% RSLogix 500 project Hourmeter.RSS, saved by version 8.30.00.16 %
PROJECT "UNTITLED"    % processor: Bul.1763 MicroLogix 1100 Series B %

PROGRAM FILES
  LAD 2   11 rungs

DATA FILES
  O0 OUTPUT  4 elements
  I1 INPUT  6 elements
  S2 STATUS  66 elements
  B3 BINARY  1 elements
  T4 TIMER  1 elements
  C5 COUNTER  3 elements
  R6 CONTROL  1 elements
  N7 INTEGER  5 elements
  F8 FLOAT  1 elements

LADDER 2
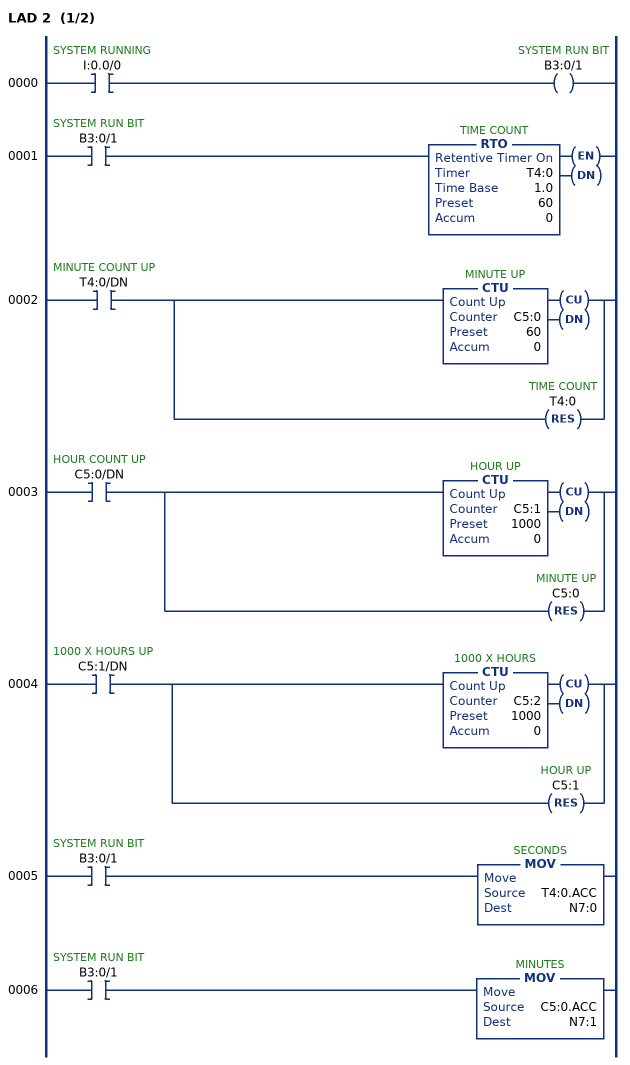
% Rung: 0 %
SOR XIC I:0.0/0 OTE B3:0/1 EOR
%   I:0.0/0  "SYSTEM RUNNING" %
%   B3:0/1  "SYSTEM RUN BIT" %
% Rung: 1 %
SOR XIC B3:0/1 RTO T4:0 1.0 60 0 EOR
%   B3:0/1  "SYSTEM RUN BIT" %
%   T4:0  "TIME COUNT" %
% Rung: 2 %
SOR XIC T4:0/DN BST CTU C5:0 60 0 NXB RES T4:0 BND EOR
%   T4:0/DN  "MINUTE COUNT UP" %
%   C5:0  "MINUTE UP" %
%   T4:0  "TIME COUNT" %
% Rung: 3 %
SOR XIC C5:0/DN BST CTU C5:1 1000 0 NXB RES C5:0 BND EOR
%   C5:0/DN  "HOUR COUNT UP" %
%   C5:1  "HOUR UP" %
%   C5:0  "MINUTE UP" %
% Rung: 4 %
SOR XIC C5:1/DN BST CTU C5:2 1000 0 NXB RES C5:1 BND EOR
%   C5:1/DN  "1000 X HOURS UP" %
%   C5:2  "1000 X HOURS" %
%   C5:1  "HOUR UP" %
% Rung: 5 %
SOR XIC B3:0/1 MOV T4:0.ACC N7:0 EOR
%   B3:0/1  "SYSTEM RUN BIT" %
%   T4:0.ACC  "SECONDS" %
%   N7:0  "SECONDS" %
% Rung: 6 %
SOR XIC B3:0/1 MOV C5:0.ACC N7:1 EOR
%   B3:0/1  "SYSTEM RUN BIT" %
%   C5:0.ACC  "MINUTES" %
%   N7:1  "MINUTES" %

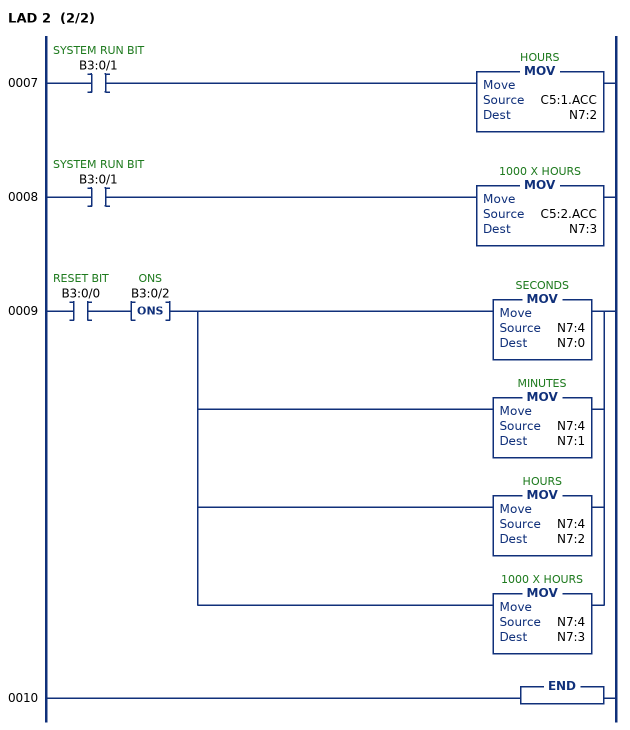
% Rung: 7 %
SOR XIC B3:0/1 MOV C5:1.ACC N7:2 EOR
%   B3:0/1  "SYSTEM RUN BIT" %
%   C5:1.ACC  "HOURS" %
%   N7:2  "HOURS" %
% Rung: 8 %
SOR XIC B3:0/1 MOV C5:2.ACC N7:3 EOR
%   B3:0/1  "SYSTEM RUN BIT" %
%   C5:2.ACC  "1000 X HOURS" %
%   N7:3  "1000 X HOURS" %
% Rung: 9 %
SOR XIC B3:0/0 ONS B3:0/2 BST MOV N7:4 N7:0 NXB BST MOV N7:4 N7:1 NXB BST MOV N7:4 N7:2 NXB MOV N7:4 N7:3 BND BND BND EOR
%   B3:0/0  "RESET BIT" %
%   B3:0/2  "ONS" %
%   N7:4  "ZERO RESET" %
%   N7:0  "SECONDS" %
%   N7:1  "MINUTES" %
%   N7:2  "HOURS" %
%   N7:3  "1000 X HOURS" %
% Rung: 10 %
SOR END EOR

OTHER DOCUMENTED ADDRESSES
  N7:0/4  "ZERO RESET"

DATA TABLE (non-zero values as saved)
DATA T4
% .PRE .ACC %
% T4:0 % 60 0
DATA C5
% .PRE .ACC %
% C5:0 % 60 0
% C5:1 % 1000 0
% C5:2 % 1000 0
